TYPE KEY_VALUE_POINTER_PAIR :
STRUCT
	Key : PVOID;
	Value : PVOID;
END_STRUCT
END_TYPE

(* stored: Version 1.1.0.1
   DUT KEY_VALUE_POINTER_PAIR: Id {8762c49f-0cec-0c19-170e-05bc9fbfd202} *)
